// TIA Portal V16 export
// export: Created 2022-11-17T15:49:47.2571168Z, ExportSetting WithDefaults, DisplayName Totally Integrated Automation Portal, DisplayVersion V16 Update 6, DisplayName TIA Portal Version Control Interface, DisplayVersion V16 Update 2, DisplayName TIA Portal Openness, DisplayVersion V16 Update 6, DisplayName SINAMICS Startdrive Advanced, DisplayVersion V16 Update 5, DisplayName SINAMICS Startdrive G130, G150, S120, S150, SINAMICS MV, S210, DisplayVersion V16 Update 5, DisplayName SINAMICS Startdrive G110M, G120, G120C, G120D, G120P, G115D, DisplayVersion V16 Update 5, DisplayName STEP 7 Professional, DisplayVersion V16 Update 6, DisplayName STEP 7 Safety, DisplayVersion V16, DisplayName WinCC Advanced, DisplayVersion V16 Update 6
DATA_BLOCK "DB320_PID"   // DB320
TITLE = PID
{ S7_Optimized_Access := 'FALSE' }
VERSION : 0.1
// stored: AutoNumber false, IsOnlyStoredInLoadMemory false, IsWriteProtectedInAS false
   VAR RETAIN
      PID { S7_SetPoint := 'True'} : "PID";
   END_VAR
BEGIN
   PID.proporzionale := 0;
   PID.integrativo := 0;
   PID.segnale := 0;
   PID.maxSegnale := 1000;
   PID.minSegnale := 0;
   PID.setPointShow := 265;
   PID.tiro := 0;
   PID.vParP := 70;
   PID.vParI := 70;
   PID.svuota := TRUE;
   PID.attiva := TRUE;
   PID.setTiro := FALSE;
   PID."timer" := T#0MS;
END_DATA_BLOCK
